{attribute 'qualified_only'}
VAR_GLOBAL
	pStringBuilder : POINTER TO CStringBuilder;
	pPara : POINTER TO ST_StringBuilderPara;
END_VAR

(* stored: Version 1.1.0.1, ProductVersion 3.1.4024.13
   GVL GVL_Strings: Id {9f669102-8e8d-43d9-8303-ff688dff9c01} *)
